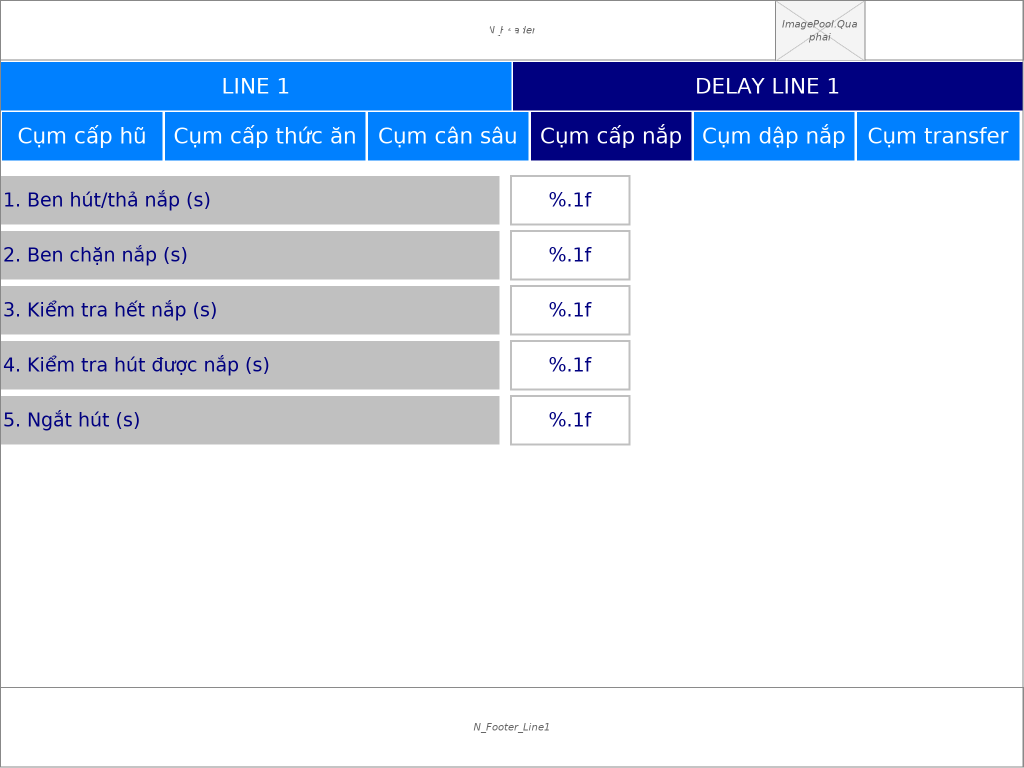
VISUALIZATION N_Setting_Delay_LidSupply1  // 1024x768
    Frame (0,687 1024x80)
        shows N_Footer_Line1()
    Frame (0,0 1024x60)
        shows N_Header()
    Textfield (353,4 420x50), "MÀN HÌNH CÀI KHOẢNG TRỄ LINE 1"
    Rectangle (0,61 512x50), "LINE 1"
        OnMouseClick: change screen: N_Setting_Line1
    Rectangle (1,111 162x50), "Cụm cấp hũ"
        OnMouseClick: change screen: N_Setting_Delay_JarSupply1
    Rectangle (164,111 202x50), "Cụm cấp thức ăn"
        OnMouseClick: change screen: N_Setting_Delay_FoodSupply1
    Rectangle (367,111 162x50), "Cụm cân sâu"
        OnMouseClick: change screen: N_Setting_Delay_WormWeight1
    Rectangle (530,111 162x50), "Cụm cấp nắp"
        OnMouseClick: change screen: N_Setting_Delay_LidSupply1
    Rectangle (693,111 162x50), "Cụm dập nắp"
        OnMouseClick: change screen: N_Setting_Delay_LidPressing1
    Rectangle (856,111 164x50), "Cụm transfer"
        OnMouseClick: change screen: N_Setting_Delay_Tranfer1
    Image (775,0 90x61), image: ImagePool.Qua phai
        OnMouseClick: change screen: N_Setting_Delay_LidSupply2
    Rectangle (0,175 500x50), "1. Ben hút/thả nắp (s)"
    Rectangle (0,230 500x50), "2. Ben chặn nắp (s)"
    Rectangle (510,175 120x50), "%.1f", text variable: PR_Line01.timerCylinder_Suction
        OnMouseClick: write PR_Line01.timerCylinder_Suction via VisuDialogs.Numpad
    Rectangle (0,285 500x50), "3. Kiểm tra hết nắp (s)"
    Rectangle (510,285 120x50), "%.1f", text variable: PR_Line01.timerCheckLidEmpty
        OnMouseClick: write PR_Line01.timerCheckLidEmpty via VisuDialogs.Numpad
    Rectangle (510,340 120x50), "%.1f", text variable: PR_Line01.timerCheckLidSuck
        OnMouseClick: write PR_Line01.timerCheckLidSuck via VisuDialogs.Numpad
    Rectangle (510,230 120x50), "%.1f", text variable: PR_Line01.timerCylinder_Stopper
        OnMouseClick: write PR_Line01.timerCylinder_Stopper via VisuDialogs.Numpad
    Rectangle (512,61 511x50), "DELAY LINE 1"
        OnMouseClick: change screen: N_Setting_Delay_JarSupply1
    Rectangle (0,340 500x50), "4. Kiểm tra hút được nắp (s)"
    Rectangle (510,395 120x50), "%.1f", text variable: PR_Line01.timerCheckLidRelease
        OnMouseClick: write PR_Line01.timerCheckLidRelease via VisuDialogs.Numpad
    Rectangle (0,395 500x50), "5. Ngắt hút (s)"
END_VISUALIZATION

(* stored: Version 1.1.0.1, ProductVersion 3.1.4024.12
   Visu N_Setting_Delay_LidSupply1: Id {453a9d8b-6126-459e-9db3-ca9bb91a0526} *)
